// TIA Portal V17 export
// export: Created 2023-01-16T15:54:28.3952353Z, ExportSetting None, DisplayName Totally Integrated Automation Portal, DisplayVersion V17, DisplayName TIA Portal Openness, DisplayVersion V17, DisplayName TIA Portal Version Control Interface, DisplayVersion V17, DisplayName STEP 7 Professional, DisplayVersion V17, DisplayName STEP 7 Safety, DisplayVersion V17, DisplayName WinCC Advanced, DisplayVersion V17
DATA_BLOCK "Data_block_1"   // DB73
{ S7_Optimized_Access := 'TRUE' }
// stored: MemoryReserve 100
BEGIN
END_DATA_BLOCK
